FUNCTION_BLOCK FB_HomingTimer
VAR_OUTPUT
	bDone : BOOL;
END_VAR
VAR
	i			: LINT := 0;
	uLoopCount	: LINT;
END_VAR


bDone := FALSE;

i := i + 1;

IF i >= uLoopCount THEN
	bDone := TRUE;
END_IF

METHOD FB_init : BOOL
VAR_INPUT
	bInitRetains	: BOOL; // if TRUE, the retain variables are initialized (warm start / cold start)
	bInCopyCode		: BOOL;  // if TRUE, the instance afterwards gets moved into the copy code (online change)
	
	uLoopsToRun		: LINT;
END_VAR

THIS^.i := 0;
THIS^.uLoopCount := uLoopsToRun;
END_METHOD

END_FUNCTION_BLOCK

(* stored: Version 1.1.0.1, ProductVersion 3.1.4024.11
   POU FB_HomingTimer: Id {6daf19c6-1dde-4928-a084-d0c6759bf0ba}, SpecialFunc None
   Method FB_init: Id {e2775d28-756d-4453-b544-630b65051fee} *)
